FUNCTION_BLOCK Q_SelectActiveWorkingSet (* Command Select Active Working Set( Part 6 - F.64 ) *)
  (* Standard: ISO 11783-6; Description: Command Select Active Working Set( Part 6 - F.64 ) This command is used by the currently active Working Set to request that the VT select a new active Working Set. This message is available in VT version 6 and later. Return values iso_s16 - E_NO_ERR - OK - E_OVERFLOW - buffer overflow - E_NOACT - Command not possible in current state - E_NO_INSTANCE - No VT client available *)
  (* Version 1.0, 2022-07-08, franz *)
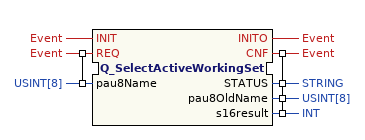
  EVENT_INPUT
    INIT; (* Service Initialization *)
    REQ WITH pau8Name; (* Service Request *)
  END_EVENT
  EVENT_OUTPUT
    INITO; (* Initialization Confirm *)
    CNF WITH STATUS, pau8OldName, s16result; (* Confirmation of Requested Service *)
  END_EVENT
  VAR_INPUT
    pau8Name : ARRAY [0..7] OF USINT; (* Iso NAME of the new active working set *)
  END_VAR
  VAR_OUTPUT
    STATUS : STRING; (* Service Status *)
    pau8OldName : ARRAY [0..7] OF USINT; (* Old value of Visible *)
    s16result : INT; (* retval see description *)
  END_VAR
END_FUNCTION_BLOCK
